// TIA Portal project "SCADA_PROJECT" (V14)

(* hardware
DEVICE "S7300/ET200M station_1"  S7-300 station
   slot 0: "Rail_0"  Rail  6ES7 390-1***0-0AA0
   slot 1: "PS 305 2A Outdoor_1"  PS 305 2A Outdoor  6ES7 305-1BA80-0AA0
   slot 2: "PLC_1"  CPU 315F-2 PN/DP  6ES7 315-2FJ14-0AB0  V3.2
      slot 2: "PROFINET interface_1"  PN-IO
         slot 1: "Port_1"  Port
         slot 2: "Port_2"  Port
   slot 4: "AI 8x12BIT_1"  AI8 x 12 bits  6ES7 331-7KF02-0AB0
   slot 5: "DO 32x24VDC/0.5A_1"  DO32 x 24VDC / 0.5A  6ES7 322-1BL00-0AA0
   slot 6: "DI 16x24VDC_1"  DI16 x 24VDC  6ES7 321-1BH50-0AA0
DEVICE "PC-System_1"  SIMATIC PC station
   slot 0: "SIMATIC PC station"  Rail  SIMATIC PC-Station  V1.0
      slot 125: "Stationmanager"  Station_Manager  V6.0.4
   slot 1: "HMI_RT_1"  WinCC RT Advanced  6AV2 104-0xxxx-xxxx  14.0.0.0
      slot 33792: "Host interface"  Host interface
   slot 2: "IE general_1"  IE General  IE_CP  V8.2.0
*)

// ===== PLC "PLC_1"  CPU 315F-2 PN/DP =====

VAR_GLOBAL   // PLC tag table "Default tag table"
   "LT1401" AT %IW256 : Int;   // Level transmitter for TANK140
   "LT1501" AT %IW258 : Int;   // Level transmitter for TANK150
   "LT1601" AT %IW260 : Int;   // Level transmitter for TANK160
   "LT1701" AT %IW262 : Int;   // Level transmitter for TANK170
   "Pump100A _start" AT %M0.0 : Bool;
   "Pump100A _stop" AT %M0.1 : Bool;
   "Pump770A _start" AT %M0.2 : Bool;
   "Pump770A_stop" AT %M0.3 : Bool;
   "Pump771A _start" AT %M0.4 : Bool;
   "Pump771A _stop" AT %M0.5 : Bool;
   "Pump100A" AT %Q4.0 : Bool;   // Status of Pump 100A
   "Pump770A" AT %Q4.1 : Bool;   // Status of Pump 770A
   "Pump771A" AT %Q4.2 : Bool;   // Status of Pump 771A
   "SV1401_open" AT %M0.6 : Bool;
   "SV1401_close" AT %M0.7 : Bool;
   "SV1501_open" AT %M1.0 : Bool;
   "SV1501_close" AT %M1.1 : Bool;
   "SV1601_open" AT %M1.2 : Bool;
   "SV1601_close" AT %M1.3 : Bool;
   "SV1701_open" AT %M1.4 : Bool;
   "SV1701_close" AT %M1.5 : Bool;
   "SV1402_open" AT %M1.6 : Bool;
   "SV1402_ close" AT %M1.7 : Bool;
   "SV1502_open" AT %M2.0 : Bool;
   "SV1502_close" AT %M2.1 : Bool;
   "SV1602_open" AT %M2.2 : Bool;
   "SV1602_ close" AT %M2.3 : Bool;
   "SV1702_open" AT %M2.4 : Bool;
   "SV1702_close" AT %M2.5 : Bool;
   "SV1401" AT %Q4.3 : Bool;   // Status of SV 1401
   "SV1501" AT %Q4.4 : Bool;   // Status of SV 1501
   "SV1601" AT %Q4.5 : Bool;   // Status of SV 1601
   "SV1701" AT %Q4.6 : Bool;   // Status of SV 1701
   "SV1402" AT %Q4.7 : Bool;   // Status of SV 1402
   "SV1502" AT %Q5.0 : Bool;   // Status of SV 1502
   "SV1602" AT %Q5.1 : Bool;   // Status of SV 1602
   "SV1702" AT %Q5.2 : Bool;   // Status of SV 1702
   "H_alarm_140" AT %Q5.3 : Bool;
   "L_alarm_140" AT %Q5.4 : Bool;
   "H_alarm_150" AT %Q5.5 : Bool;
   "L_alarm_150" AT %Q5.6 : Bool;
   "H_alarm_160" AT %Q5.7 : Bool;
   "L_alarm_160" AT %Q6.0 : Bool;
   "H_alarm_170" AT %Q6.1 : Bool;
   "L_alarm_170" AT %Q6.2 : Bool;
   "Level_real_140" AT %MD6 : Real;   // Analog value for level in Tank 140
   "Level_real_150" AT %MD10 : Real;   // Analog value for level in Tank 150
   "Level_real_160" AT %MD14 : Real;   // Analog value for level in Tank 160
   "Level_real_170" AT %MD18 : Real;   // Analog value for level in Tank 170
   "Tag_2" AT %M3.0 : Bool;   // LT140 incoming alarm
   "Tag_3" AT %M3.1 : Bool;   // LT140 out of alarm
   "Tag_4" AT %M3.2 : Bool;   // LT150 incoming alarm
   "Tag_6" AT %M3.4 : Bool;   // Pump 771A incoming alarm
   "Tag_8" AT %M3.6 : Bool;   // Pump 771A out of alarm
   "Tag_7" AT %M3.5 : Bool;   // SV1401 incoming alarm
   "Tag_9" AT %M3.7 : Bool;   // SV1401 out of alarm
   "Tag_5" AT %M3.3 : Bool;   // LT140 out of alarm
END_VAR

VAR_GLOBAL CONSTANT   // PLC tag table "Default tag table"
   "MAX_level_140" : Real := 1500.0;
   "MIN_level_140" : Real := 0.0;
   "HIGH_level_140" : Real := 1350.0;
   "LOW_level_140" : Real := 200.0;
   "MAX_level_150" : Real := 2500.0;
   "MIN_level_150" : Real := 0.0;
   "HIGH_level_150" : Real := 2250.0;
   "LOW_level_150" : Real := 200.0;
   "MAX_level_160" : Real := 3000.0;
   "MIN_level_160" : Real := 0.0;
   "HIGH_level_160" : Real := 2700.0;
   "LOW_level_160" : Real := 200.0;
   "MAX_level_170" : Real := 10000.0;
   "MIN_level_170" : Real := 0.0;
   "HIGH_level_170" : Real := 9000.0;
   "LOW_level_170" : Real := 1000.0;
END_VAR

DATA_BLOCK "FP_Database"   // DB1
{ S7_Optimized_Access := 'FALSE' }
VERSION : 0.1
   VAR
      Pump_visibility_1 : Bool := false;
      Pump100A : String := 'Pump100A';
      Pump_visibility_2 : Bool := false;
      Pump770 : String := 'Pump770';
      Pump_visibility_3 : Bool := false;
      Pump771 : String := 'Pump771';
      V_vis_1401 : Bool := false;
      "SV 1401" : String := 'SV 1401';
      V_vis_1501 : Bool := false;
      SV1501 : String := 'SV 1501';
      V_vis_1601 : Bool := false;
      SV1601 : String := 'SV 1601';
      V_vis_1701 : Bool := false;
      SV1701 : String := 'SV 1701';
      V_vis_1402 : Bool := false;
      SV1402 : String := 'SV 1402';
      V_vis_1502 : Bool := false;
      SV1502 : String := 'SV 1502';
      V_vis_1602 : Bool := false;
      SV1602 : String := 'SV 1602';
      V_vis_1702 : Bool := false;
      SV1702 : String := 'SV 1702';
   END_VAR
BEGIN
END_DATA_BLOCK

DATA_BLOCK "Alarm_DB"   // DB2
{ S7_Optimized_Access := 'FALSE' }
VERSION : 0.1
   VAR
      LT140_fault : Bool;
      LT150_fault : Bool;
      SV1401_FTC : Bool;
      SV1502_FTO : Bool;
      Pump771_FTS : Bool;
   END_VAR
BEGIN
END_DATA_BLOCK

FUNCTION "SV1x01" : Void   // FC1, LAD
{ S7_Optimized_Access := 'FALSE' }
VERSION : 0.1
   VAR_INPUT
      Open_valve : Bool;
      close_valve : Bool;
      High_alarm : Bool;
      Stop_pump : Bool;
      "Low alarm" : Bool;
   END_VAR
   VAR_OUTPUT
      SV1x01 : Bool;
   END_VAR
BEGIN

REGION Network 1
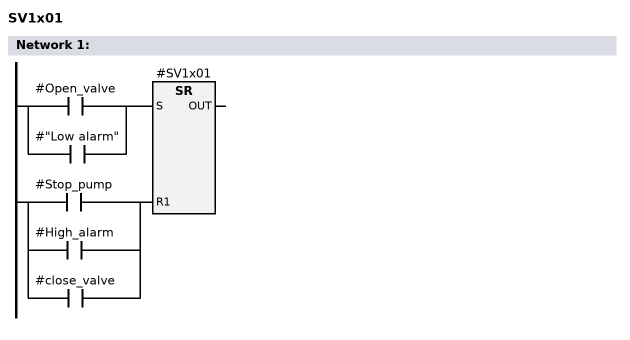
   RUNG wire#powerrail
      Contact( #Open_valve )
      wire#w1
      S_SR(operand := #SV1x01, r1 := wire#w2)
   END_RUNG
   RUNG wire#powerrail
      Contact( #"Low alarm" )
   END_RUNG wire#w1
   RUNG wire#powerrail
      Contact( #Stop_pump )
   END_RUNG wire#w2
   RUNG wire#powerrail
      Contact( #High_alarm )
   END_RUNG wire#w2
   RUNG wire#powerrail
      Contact( #close_valve )
   END_RUNG wire#w2
   // the same network as SCL:
   IF #Open_valve OR #"Low alarm" THEN
       #SV1x01 := TRUE;   // SR flip-flop
   END_IF;
   IF #Stop_pump OR #High_alarm OR #close_valve THEN #SV1x01 := FALSE; END_IF;
END_REGION
END_FUNCTION

FUNCTION "Tank_Alarm" : Void   // FC2, LAD
{ S7_Optimized_Access := 'FALSE' }
VERSION : 0.1
   VAR_INPUT
      LT1x01 : Int;
      High_Level : Real;
      Low_Level : Real;
      HIGH_alarm_limit : Real;
      LOW_alarm_limit : Real;
   END_VAR
   VAR_OUTPUT
      High_alarm : Bool;
      Low_alarm : Bool;
   END_VAR
   VAR_IN_OUT
      Level : Real;
   END_VAR
   VAR_TEMP
      Bipolar : Bool;
      Value : Word;
   END_VAR
BEGIN

REGION Network 1
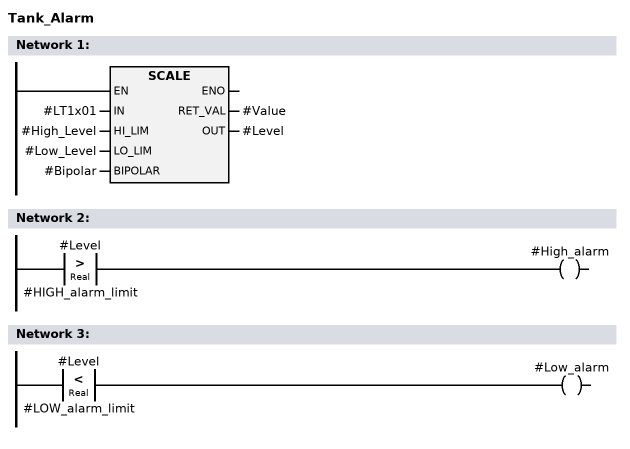
   #Value := SCALE(IN := #LT1x01,
                   HI_LIM := #High_Level,
                   LO_LIM := #Low_Level,
                   BIPOLAR := #Bipolar,
                   OUT => #Level);
END_REGION

REGION Network 2
   RUNG wire#powerrail
      { S7_Templates := "SrcType := Real" } GT_Contact(in1 := #Level, in2 := #HIGH_alarm_limit)
      Coil( #High_alarm )
   END_RUNG
   // the same network as SCL:
   #High_alarm := #Level > #HIGH_alarm_limit;
END_REGION

REGION Network 3
   RUNG wire#powerrail
      { S7_Templates := "SrcType := Real" } LT_Contact(in1 := #Level, in2 := #LOW_alarm_limit)
      Coil( #Low_alarm )
   END_RUNG
   // the same network as SCL:
   #Low_alarm := #Level < #LOW_alarm_limit;
END_REGION
END_FUNCTION

FUNCTION "PUMP_100A" : Void   // FC3, LAD
{ S7_Optimized_Access := 'FALSE' }
VERSION : 0.1
   VAR_INPUT
      SV1x01_1 : Bool;
      SVx01_2 : Bool;
      SV1x01_3 : Bool;
      START_PUMP : Bool;
      STOP_PUMP : Bool;
      Pump770A : Bool;
      SV1701 : Bool;
      L_140 : Bool;
      L_150 : Bool;
      L_160 : Bool;
   END_VAR
   VAR_OUTPUT
      PUMP100A : Bool;
   END_VAR
BEGIN

REGION Network 1
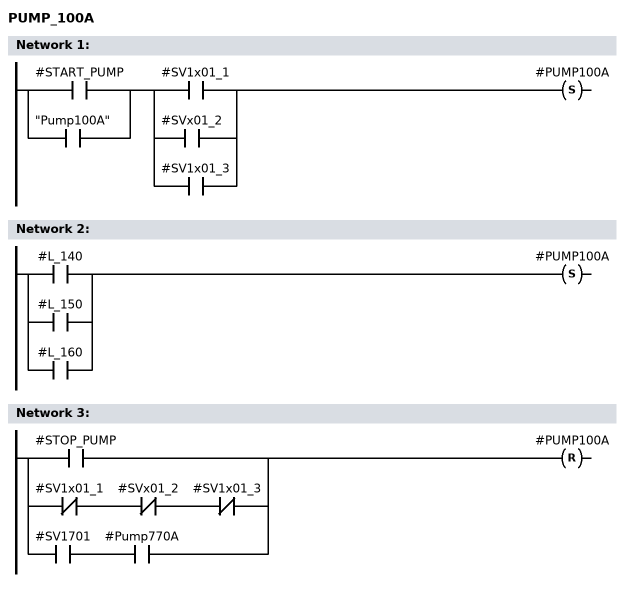
   RUNG wire#powerrail
      Contact( #START_PUMP )
      wire#w1
      Contact( #SV1x01_1 )
      wire#w2
      S_Coil( #PUMP100A )
   END_RUNG
   RUNG wire#powerrail
      Contact( "Pump100A" )
   END_RUNG wire#w1
   RUNG wire#w1
      Contact( #SVx01_2 )
   END_RUNG wire#w2
   RUNG wire#w1
      Contact( #SV1x01_3 )
   END_RUNG wire#w2
   // the same network as SCL:
   IF (#START_PUMP OR "Pump100A") AND (#SV1x01_1 OR #SVx01_2 OR #SV1x01_3) THEN #PUMP100A := TRUE; END_IF;
END_REGION

REGION Network 2
   RUNG wire#powerrail
      Contact( #L_140 )
      wire#w1
      S_Coil( #PUMP100A )
   END_RUNG
   RUNG wire#powerrail
      Contact( #L_150 )
   END_RUNG wire#w1
   RUNG wire#powerrail
      Contact( #L_160 )
   END_RUNG wire#w1
   // the same network as SCL:
   IF #L_140 OR #L_150 OR #L_160 THEN #PUMP100A := TRUE; END_IF;
END_REGION

REGION Network 3
   RUNG wire#powerrail
      Contact( #STOP_PUMP )
      wire#w1
      R_Coil( #PUMP100A )
   END_RUNG
   RUNG wire#powerrail
      I_Contact( #SV1x01_1 )
      I_Contact( #SVx01_2 )
      I_Contact( #SV1x01_3 )
   END_RUNG wire#w1
   RUNG wire#powerrail
      Contact( #SV1701 )
      Contact( #Pump770A )
   END_RUNG wire#w1
   // the same network as SCL:
   IF #STOP_PUMP OR (NOT #SV1x01_1 AND NOT #SVx01_2 AND NOT #SV1x01_3) OR (#SV1701 AND #Pump770A) THEN
       #PUMP100A := FALSE;
   END_IF;
END_REGION
END_FUNCTION

FUNCTION "SV1x02" : Void   // FC4, LAD
{ S7_Optimized_Access := 'FALSE' }
VERSION : 0.1
   VAR_INPUT
      Open_valve : Bool;
      SV1x01 : Bool;
      Low_alarm_170 : Bool;
      High_Alarm : Bool;
      Low_alarm : Bool;
      High_alarm_170 : Bool;
      close_valve : Bool;
      Pump100A : Bool;
   END_VAR
   VAR_OUTPUT
      SV_1x02 : Bool;
   END_VAR
BEGIN

REGION Network 1
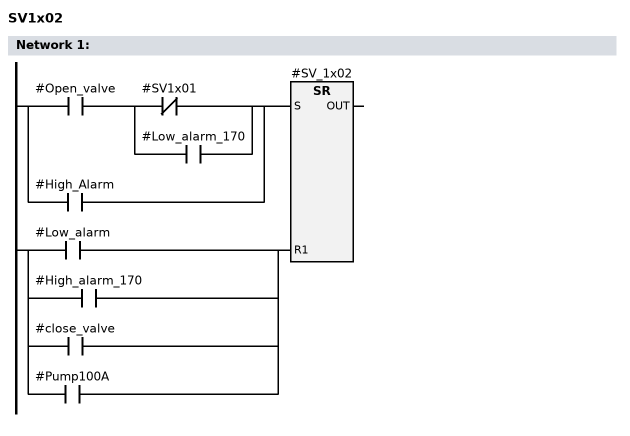
   RUNG wire#powerrail
      Contact( #Open_valve )
      wire#w1
      I_Contact( #SV1x01 )
      wire#w2
      S_SR(operand := #SV_1x02, r1 := wire#w3)
   END_RUNG
   RUNG wire#w1
      Contact( #Low_alarm_170 )
   END_RUNG wire#w2
   RUNG wire#powerrail
      Contact( #High_Alarm )
   END_RUNG wire#w2
   RUNG wire#powerrail
      Contact( #Low_alarm )
   END_RUNG wire#w3
   RUNG wire#powerrail
      Contact( #High_alarm_170 )
   END_RUNG wire#w3
   RUNG wire#powerrail
      Contact( #close_valve )
   END_RUNG wire#w3
   RUNG wire#powerrail
      Contact( #Pump100A )
   END_RUNG wire#w3
   // the same network as SCL:
   IF (#Open_valve AND (NOT #SV1x01 OR #Low_alarm_170)) OR #High_Alarm THEN
       #SV_1x02 := TRUE;   // SR flip-flop
   END_IF;
   IF #Low_alarm OR #High_alarm_170 OR #close_valve OR #Pump100A THEN #SV_1x02 := FALSE; END_IF;
END_REGION
END_FUNCTION

FUNCTION "SV_1702" : Void   // FC6, LAD
{ S7_Optimized_Access := 'FALSE' }
VERSION : 0.1
   VAR_INPUT
      Open_valve : Bool;
      High_170 : Bool;
      Close_valve : Bool;
      LOW_170 : Bool;
      SV1701 : Bool;
      PUMP770A : Bool;
   END_VAR
   VAR_OUTPUT
      SV_1702 : Bool;
   END_VAR
BEGIN

REGION Network 1
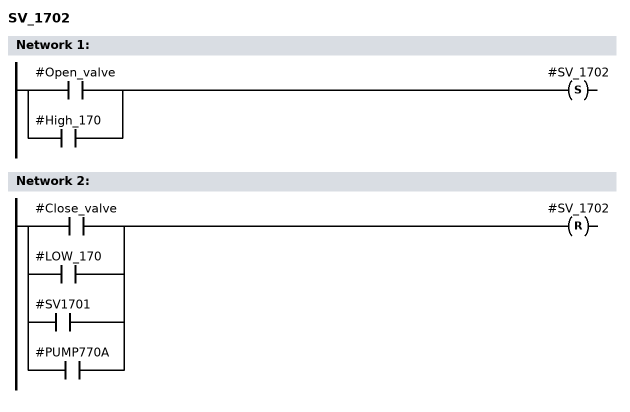
   RUNG wire#powerrail
      Contact( #Open_valve )
      wire#w1
      S_Coil( #SV_1702 )
   END_RUNG
   RUNG wire#powerrail
      Contact( #High_170 )
   END_RUNG wire#w1
   // the same network as SCL:
   IF #Open_valve OR #High_170 THEN #SV_1702 := TRUE; END_IF;
END_REGION

REGION Network 2
   RUNG wire#powerrail
      Contact( #Close_valve )
      wire#w1
      R_Coil( #SV_1702 )
   END_RUNG
   RUNG wire#powerrail
      Contact( #LOW_170 )
   END_RUNG wire#w1
   RUNG wire#powerrail
      Contact( #SV1701 )
   END_RUNG wire#w1
   RUNG wire#powerrail
      Contact( #PUMP770A )
   END_RUNG wire#w1
   // the same network as SCL:
   IF #Close_valve OR #LOW_170 OR #SV1701 OR #PUMP770A THEN #SV_1702 := FALSE; END_IF;
END_REGION
END_FUNCTION

FUNCTION "PUMP_770A" : Void   // FC7, LAD
{ S7_Optimized_Access := 'FALSE' }
VERSION : 0.1
   VAR_INPUT
      Start_pump : Bool;
      SV1701 : Bool;
      Low170 : Bool;
      Stop_pump : Bool;
      High170 : Bool;
      SV1x02_1 : Bool;
      SVx02_2 : Bool;
      SV1x02_3 : Bool;
      SV1702 : Bool;
      "PUMP _771A" : Bool;
      PUMP_100A : Bool;
   END_VAR
   VAR_OUTPUT
      Pump770 : Bool;
   END_VAR
BEGIN

REGION Network 1
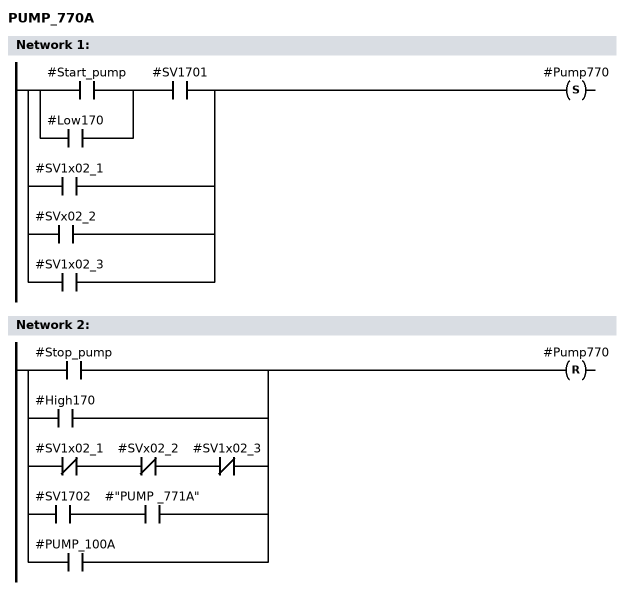
   RUNG wire#powerrail
      Contact( #Start_pump )
      wire#w1
      Contact( #SV1701 )
      wire#w2
      S_Coil( #Pump770 )
   END_RUNG
   RUNG wire#powerrail
      Contact( #Low170 )
   END_RUNG wire#w1
   RUNG wire#powerrail
      Contact( #SV1x02_1 )
   END_RUNG wire#w2
   RUNG wire#powerrail
      Contact( #SVx02_2 )
   END_RUNG wire#w2
   RUNG wire#powerrail
      Contact( #SV1x02_3 )
   END_RUNG wire#w2
   // the same network as SCL:
   IF ((#Start_pump OR #Low170) AND #SV1701) OR #SV1x02_1 OR #SVx02_2 OR #SV1x02_3 THEN
       #Pump770 := TRUE;
   END_IF;
END_REGION

REGION Network 2
   RUNG wire#powerrail
      Contact( #Stop_pump )
      wire#w1
      R_Coil( #Pump770 )
   END_RUNG
   RUNG wire#powerrail
      Contact( #High170 )
   END_RUNG wire#w1
   RUNG wire#powerrail
      I_Contact( #SV1x02_1 )
      I_Contact( #SVx02_2 )
      I_Contact( #SV1x02_3 )
   END_RUNG wire#w1
   RUNG wire#powerrail
      Contact( #SV1702 )
      Contact( #"PUMP _771A" )
   END_RUNG wire#w1
   RUNG wire#powerrail
      Contact( #PUMP_100A )
   END_RUNG wire#w1
   // the same network as SCL:
   IF #Stop_pump OR #High170 OR (NOT #SV1x02_1 AND NOT #SVx02_2 AND NOT #SV1x02_3) OR (#SV1702 AND #"PUMP _771A") OR #PUMP_100A THEN
       #Pump770 := FALSE;
   END_IF;
END_REGION
END_FUNCTION

FUNCTION "PUMP_771A" : Void   // FC8, LAD
{ S7_Optimized_Access := 'FALSE' }
VERSION : 0.1
   VAR_INPUT
      START_PUMP : Bool;
      SV1702 : Bool;
      High_170 : Bool;
      STOP_Pump : Bool;
      LOW_170 : Bool;
      SV1701 : Bool;
      Pump770A : Bool;
      Pump100A : Bool;
   END_VAR
   VAR_OUTPUT
      PUMP771A : Bool;
   END_VAR
BEGIN

REGION Network 1
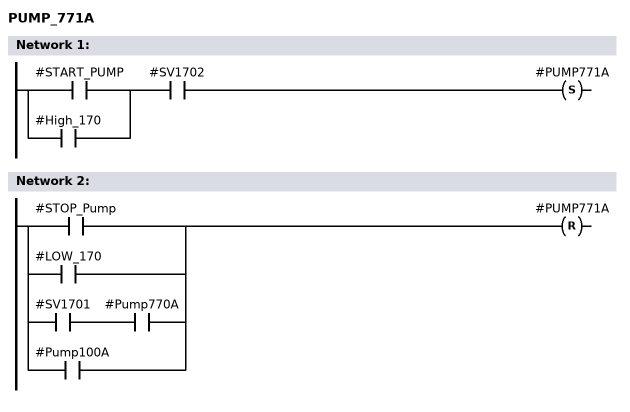
   RUNG wire#powerrail
      Contact( #START_PUMP )
      wire#w1
      Contact( #SV1702 )
      S_Coil( #PUMP771A )
   END_RUNG
   RUNG wire#powerrail
      Contact( #High_170 )
   END_RUNG wire#w1
   // the same network as SCL:
   IF (#START_PUMP OR #High_170) AND #SV1702 THEN #PUMP771A := TRUE; END_IF;
END_REGION

REGION Network 2
   RUNG wire#powerrail
      Contact( #STOP_Pump )
      wire#w1
      R_Coil( #PUMP771A )
   END_RUNG
   RUNG wire#powerrail
      Contact( #LOW_170 )
   END_RUNG wire#w1
   RUNG wire#powerrail
      Contact( #SV1701 )
      Contact( #Pump770A )
   END_RUNG wire#w1
   RUNG wire#powerrail
      Contact( #Pump100A )
   END_RUNG wire#w1
   // the same network as SCL:
   IF #STOP_Pump OR #LOW_170 OR (#SV1701 AND #Pump770A) OR #Pump100A THEN #PUMP771A := FALSE; END_IF;
END_REGION
END_FUNCTION

FUNCTION "SV_1701" : Void   // FC9, LAD
{ S7_Optimized_Access := 'FALSE' }
VERSION : 0.1
   VAR_INPUT
      OPEN_valve : Bool;
      SV1402 : Bool;
      SV1502 : Bool;
      SV1602 : Bool;
      Close_valve : Bool;
      HIGH_170 : Bool;
   END_VAR
   VAR_OUTPUT
      SV1701 : Bool;
   END_VAR
BEGIN

REGION Network 1
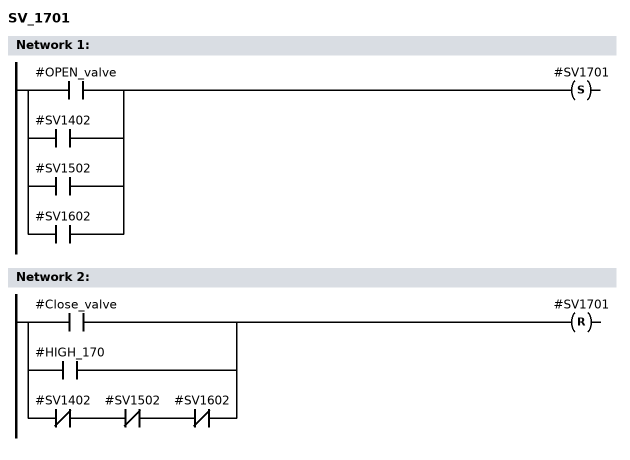
   RUNG wire#powerrail
      Contact( #OPEN_valve )
      wire#w1
      S_Coil( #SV1701 )
   END_RUNG
   RUNG wire#powerrail
      Contact( #SV1402 )
   END_RUNG wire#w1
   RUNG wire#powerrail
      Contact( #SV1502 )
   END_RUNG wire#w1
   RUNG wire#powerrail
      Contact( #SV1602 )
   END_RUNG wire#w1
   // the same network as SCL:
   IF #OPEN_valve OR #SV1402 OR #SV1502 OR #SV1602 THEN #SV1701 := TRUE; END_IF;
END_REGION

REGION Network 2
   RUNG wire#powerrail
      Contact( #Close_valve )
      wire#w1
      R_Coil( #SV1701 )
   END_RUNG
   RUNG wire#powerrail
      Contact( #HIGH_170 )
   END_RUNG wire#w1
   RUNG wire#powerrail
      I_Contact( #SV1402 )
      I_Contact( #SV1502 )
      I_Contact( #SV1602 )
   END_RUNG wire#w1
   // the same network as SCL:
   IF #Close_valve OR #HIGH_170 OR (NOT #SV1402 AND NOT #SV1502 AND NOT #SV1602) THEN
       #SV1701 := FALSE;
   END_IF;
END_REGION
END_FUNCTION

ORGANIZATION_BLOCK "Main"   // OB1, LAD
TITLE = "Main Program Sweep (Cycle)"
{ S7_Optimized_Access := 'FALSE' }
VERSION : 0.1
   VAR_TEMP
      OB1_EV_CLASS : Byte;   // Bits 0-3 = 1 (Coming event), Bits 4-7 = 1 (Event class 1)
      OB1_SCAN_1 : Byte;   // 1 (Cold restart scan 1 of OB 1), 3 (Scan 2-n of OB 1)
      OB1_PRIORITY : Byte;   // Priority of OB Execution
      OB1_OB_NUMBR : Byte;   // 1 (Organization block 1, OB1)
      OB1_RESERVED_1 : Byte;   // Reserved for system
      OB1_RESERVED_2 : Byte;   // Reserved for system
      OB1_PREV_CYCLE : Int;   // Cycle time of previous OB1 scan (milliseconds)
      OB1_MIN_CYCLE : Int;   // Minimum cycle time of OB1 (milliseconds)
      OB1_MAX_CYCLE : Int;   // Maximum cycle time of OB1 (milliseconds)
      OB1_DATE_TIME : Date_And_Time;   // Date and time OB1 started
   END_VAR
BEGIN

REGION Network 1
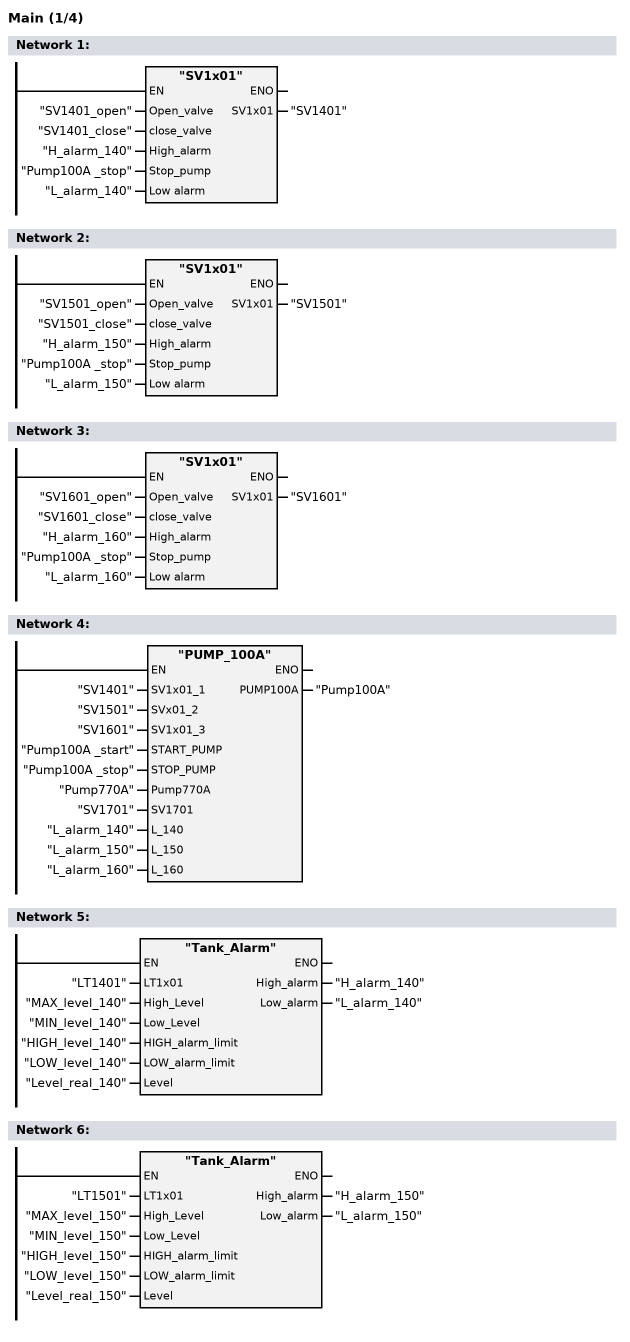
   RUNG wire#powerrail
      "SV1x01"(Open_valve := "SV1401_open", close_valve := "SV1401_close", High_alarm := "H_alarm_140", Stop_pump := "Pump100A _stop", "Low alarm" := "L_alarm_140", SV1x01 => "SV1401")
   END_RUNG
   // the same network as SCL:
   "SV1x01"(Open_valve := "SV1401_open",
            close_valve := "SV1401_close",
            High_alarm := "H_alarm_140",
            Stop_pump := "Pump100A _stop",
            "Low alarm" := "L_alarm_140",
            SV1x01 => "SV1401");
END_REGION

REGION Network 2
   RUNG wire#powerrail
      "SV1x01"(Open_valve := "SV1501_open", close_valve := "SV1501_close", High_alarm := "H_alarm_150", Stop_pump := "Pump100A _stop", "Low alarm" := "L_alarm_150", SV1x01 => "SV1501")
   END_RUNG
   // the same network as SCL:
   "SV1x01"(Open_valve := "SV1501_open",
            close_valve := "SV1501_close",
            High_alarm := "H_alarm_150",
            Stop_pump := "Pump100A _stop",
            "Low alarm" := "L_alarm_150",
            SV1x01 => "SV1501");
END_REGION

REGION Network 3
   RUNG wire#powerrail
      "SV1x01"(Open_valve := "SV1601_open", close_valve := "SV1601_close", High_alarm := "H_alarm_160", Stop_pump := "Pump100A _stop", "Low alarm" := "L_alarm_160", SV1x01 => "SV1601")
   END_RUNG
   // the same network as SCL:
   "SV1x01"(Open_valve := "SV1601_open",
            close_valve := "SV1601_close",
            High_alarm := "H_alarm_160",
            Stop_pump := "Pump100A _stop",
            "Low alarm" := "L_alarm_160",
            SV1x01 => "SV1601");
END_REGION

REGION Network 4
   RUNG wire#powerrail
      "PUMP_100A"(SV1x01_1 := "SV1401", SVx01_2 := "SV1501", SV1x01_3 := "SV1601", START_PUMP := "Pump100A _start", STOP_PUMP := "Pump100A _stop", Pump770A := "Pump770A", SV1701 := "SV1701", L_140 := "L_alarm_140", L_150 := "L_alarm_150", L_160 := "L_alarm_160", PUMP100A => "Pump100A")
   END_RUNG
   // the same network as SCL:
   "PUMP_100A"(SV1x01_1 := "SV1401",
               SVx01_2 := "SV1501",
               SV1x01_3 := "SV1601",
               START_PUMP := "Pump100A _start",
               STOP_PUMP := "Pump100A _stop",
               Pump770A := "Pump770A",
               SV1701 := "SV1701",
               L_140 := "L_alarm_140",
               L_150 := "L_alarm_150",
               L_160 := "L_alarm_160",
               PUMP100A => "Pump100A");
END_REGION

REGION Network 5
   RUNG wire#powerrail
      "Tank_Alarm"(LT1x01 := "LT1401", High_Level := "MAX_level_140", Low_Level := "MIN_level_140", HIGH_alarm_limit := "HIGH_level_140", LOW_alarm_limit := "LOW_level_140", Level := "Level_real_140", High_alarm => "H_alarm_140", Low_alarm => "L_alarm_140")
   END_RUNG
   // the same network as SCL:
   "Tank_Alarm"(LT1x01 := "LT1401",
                High_Level := "MAX_level_140",
                Low_Level := "MIN_level_140",
                HIGH_alarm_limit := "HIGH_level_140",
                LOW_alarm_limit := "LOW_level_140",
                Level := "Level_real_140",
                High_alarm => "H_alarm_140",
                Low_alarm => "L_alarm_140");
END_REGION

REGION Network 6
   RUNG wire#powerrail
      "Tank_Alarm"(LT1x01 := "LT1501", High_Level := "MAX_level_150", Low_Level := "MIN_level_150", HIGH_alarm_limit := "HIGH_level_150", LOW_alarm_limit := "LOW_level_150", Level := "Level_real_150", High_alarm => "H_alarm_150", Low_alarm => "L_alarm_150")
   END_RUNG
   // the same network as SCL:
   "Tank_Alarm"(LT1x01 := "LT1501",
                High_Level := "MAX_level_150",
                Low_Level := "MIN_level_150",
                HIGH_alarm_limit := "HIGH_level_150",
                LOW_alarm_limit := "LOW_level_150",
                Level := "Level_real_150",
                High_alarm => "H_alarm_150",
                Low_alarm => "L_alarm_150");
END_REGION

REGION Network 7
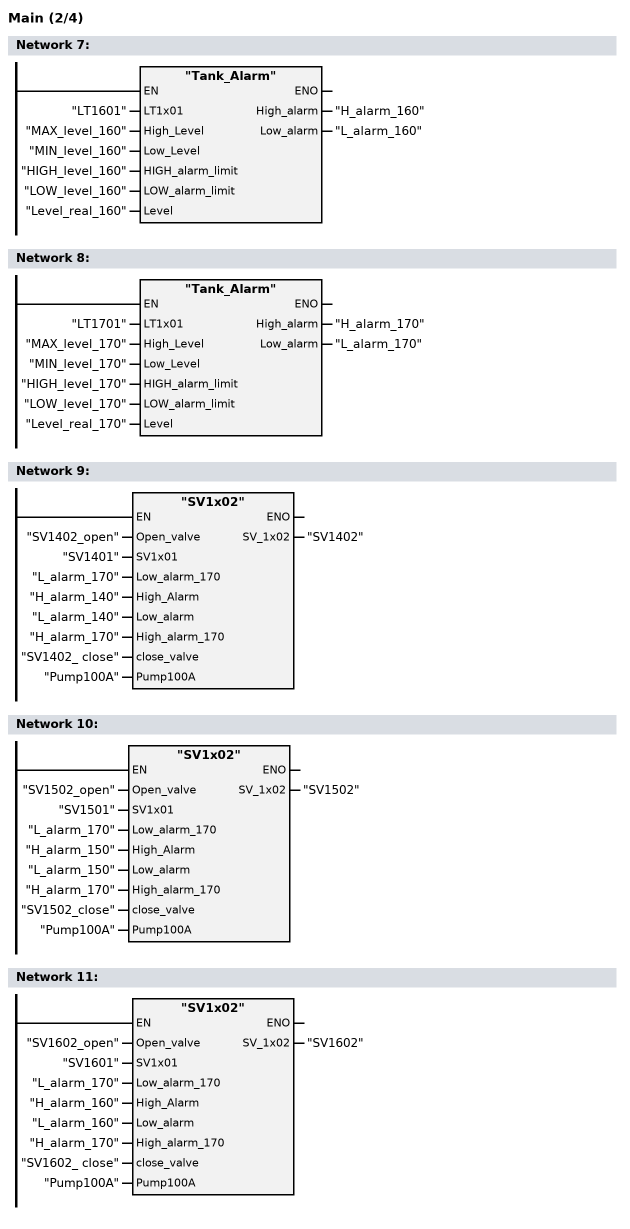
   RUNG wire#powerrail
      "Tank_Alarm"(LT1x01 := "LT1601", High_Level := "MAX_level_160", Low_Level := "MIN_level_160", HIGH_alarm_limit := "HIGH_level_160", LOW_alarm_limit := "LOW_level_160", Level := "Level_real_160", High_alarm => "H_alarm_160", Low_alarm => "L_alarm_160")
   END_RUNG
   // the same network as SCL:
   "Tank_Alarm"(LT1x01 := "LT1601",
                High_Level := "MAX_level_160",
                Low_Level := "MIN_level_160",
                HIGH_alarm_limit := "HIGH_level_160",
                LOW_alarm_limit := "LOW_level_160",
                Level := "Level_real_160",
                High_alarm => "H_alarm_160",
                Low_alarm => "L_alarm_160");
END_REGION

REGION Network 8
   RUNG wire#powerrail
      "Tank_Alarm"(LT1x01 := "LT1701", High_Level := "MAX_level_170", Low_Level := "MIN_level_170", HIGH_alarm_limit := "HIGH_level_170", LOW_alarm_limit := "LOW_level_170", Level := "Level_real_170", High_alarm => "H_alarm_170", Low_alarm => "L_alarm_170")
   END_RUNG
   // the same network as SCL:
   "Tank_Alarm"(LT1x01 := "LT1701",
                High_Level := "MAX_level_170",
                Low_Level := "MIN_level_170",
                HIGH_alarm_limit := "HIGH_level_170",
                LOW_alarm_limit := "LOW_level_170",
                Level := "Level_real_170",
                High_alarm => "H_alarm_170",
                Low_alarm => "L_alarm_170");
END_REGION

REGION Network 9
   RUNG wire#powerrail
      "SV1x02"(Open_valve := "SV1402_open", SV1x01 := "SV1401", Low_alarm_170 := "L_alarm_170", High_Alarm := "H_alarm_140", Low_alarm := "L_alarm_140", High_alarm_170 := "H_alarm_170", close_valve := "SV1402_ close", Pump100A := "Pump100A", SV_1x02 => "SV1402")
   END_RUNG
   // the same network as SCL:
   "SV1x02"(Open_valve := "SV1402_open",
            SV1x01 := "SV1401",
            Low_alarm_170 := "L_alarm_170",
            High_Alarm := "H_alarm_140",
            Low_alarm := "L_alarm_140",
            High_alarm_170 := "H_alarm_170",
            close_valve := "SV1402_ close",
            Pump100A := "Pump100A",
            SV_1x02 => "SV1402");
END_REGION

REGION Network 10
   RUNG wire#powerrail
      "SV1x02"(Open_valve := "SV1502_open", SV1x01 := "SV1501", Low_alarm_170 := "L_alarm_170", High_Alarm := "H_alarm_150", Low_alarm := "L_alarm_150", High_alarm_170 := "H_alarm_170", close_valve := "SV1502_close", Pump100A := "Pump100A", SV_1x02 => "SV1502")
   END_RUNG
   // the same network as SCL:
   "SV1x02"(Open_valve := "SV1502_open",
            SV1x01 := "SV1501",
            Low_alarm_170 := "L_alarm_170",
            High_Alarm := "H_alarm_150",
            Low_alarm := "L_alarm_150",
            High_alarm_170 := "H_alarm_170",
            close_valve := "SV1502_close",
            Pump100A := "Pump100A",
            SV_1x02 => "SV1502");
END_REGION

REGION Network 11
   RUNG wire#powerrail
      "SV1x02"(Open_valve := "SV1602_open", SV1x01 := "SV1601", Low_alarm_170 := "L_alarm_170", High_Alarm := "H_alarm_160", Low_alarm := "L_alarm_160", High_alarm_170 := "H_alarm_170", close_valve := "SV1602_ close", Pump100A := "Pump100A", SV_1x02 => "SV1602")
   END_RUNG
   // the same network as SCL:
   "SV1x02"(Open_valve := "SV1602_open",
            SV1x01 := "SV1601",
            Low_alarm_170 := "L_alarm_170",
            High_Alarm := "H_alarm_160",
            Low_alarm := "L_alarm_160",
            High_alarm_170 := "H_alarm_170",
            close_valve := "SV1602_ close",
            Pump100A := "Pump100A",
            SV_1x02 => "SV1602");
END_REGION

REGION Network 12
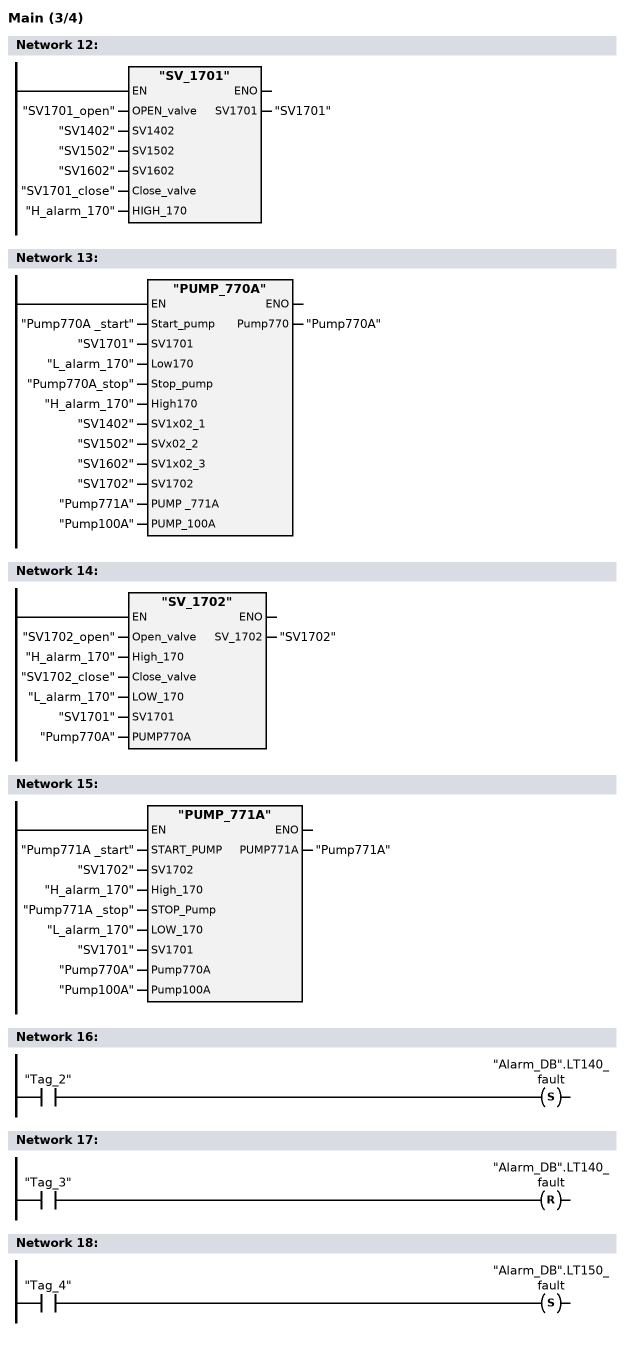
   RUNG wire#powerrail
      "SV_1701"(OPEN_valve := "SV1701_open", SV1402 := "SV1402", SV1502 := "SV1502", SV1602 := "SV1602", Close_valve := "SV1701_close", HIGH_170 := "H_alarm_170", SV1701 => "SV1701")
   END_RUNG
   // the same network as SCL:
   "SV_1701"(OPEN_valve := "SV1701_open",
             SV1402 := "SV1402",
             SV1502 := "SV1502",
             SV1602 := "SV1602",
             Close_valve := "SV1701_close",
             HIGH_170 := "H_alarm_170",
             SV1701 => "SV1701");
END_REGION

REGION Network 13
   RUNG wire#powerrail
      "PUMP_770A"(Start_pump := "Pump770A _start", SV1701 := "SV1701", Low170 := "L_alarm_170", Stop_pump := "Pump770A_stop", High170 := "H_alarm_170", SV1x02_1 := "SV1402", SVx02_2 := "SV1502", SV1x02_3 := "SV1602", SV1702 := "SV1702", "PUMP _771A" := "Pump771A", PUMP_100A := "Pump100A", Pump770 => "Pump770A")
   END_RUNG
   // the same network as SCL:
   "PUMP_770A"(Start_pump := "Pump770A _start",
               SV1701 := "SV1701",
               Low170 := "L_alarm_170",
               Stop_pump := "Pump770A_stop",
               High170 := "H_alarm_170",
               SV1x02_1 := "SV1402",
               SVx02_2 := "SV1502",
               SV1x02_3 := "SV1602",
               SV1702 := "SV1702",
               "PUMP _771A" := "Pump771A",
               PUMP_100A := "Pump100A",
               Pump770 => "Pump770A");
END_REGION

REGION Network 14
   RUNG wire#powerrail
      "SV_1702"(Open_valve := "SV1702_open", High_170 := "H_alarm_170", Close_valve := "SV1702_close", LOW_170 := "L_alarm_170", SV1701 := "SV1701", PUMP770A := "Pump770A", SV_1702 => "SV1702")
   END_RUNG
   // the same network as SCL:
   "SV_1702"(Open_valve := "SV1702_open",
             High_170 := "H_alarm_170",
             Close_valve := "SV1702_close",
             LOW_170 := "L_alarm_170",
             SV1701 := "SV1701",
             PUMP770A := "Pump770A",
             SV_1702 => "SV1702");
END_REGION

REGION Network 15
   RUNG wire#powerrail
      "PUMP_771A"(START_PUMP := "Pump771A _start", SV1702 := "SV1702", High_170 := "H_alarm_170", STOP_Pump := "Pump771A _stop", LOW_170 := "L_alarm_170", SV1701 := "SV1701", Pump770A := "Pump770A", Pump100A := "Pump100A", PUMP771A => "Pump771A")
   END_RUNG
   // the same network as SCL:
   "PUMP_771A"(START_PUMP := "Pump771A _start",
               SV1702 := "SV1702",
               High_170 := "H_alarm_170",
               STOP_Pump := "Pump771A _stop",
               LOW_170 := "L_alarm_170",
               SV1701 := "SV1701",
               Pump770A := "Pump770A",
               Pump100A := "Pump100A",
               PUMP771A => "Pump771A");
END_REGION

REGION Network 16
   RUNG wire#powerrail
      Contact( "Tag_2" )
      S_Coil( "Alarm_DB".LT140_fault )
   END_RUNG
   // the same network as SCL:
   IF "Tag_2" THEN "Alarm_DB".LT140_fault := TRUE; END_IF;
END_REGION

REGION Network 17
   RUNG wire#powerrail
      Contact( "Tag_3" )
      R_Coil( "Alarm_DB".LT140_fault )
   END_RUNG
   // the same network as SCL:
   IF "Tag_3" THEN "Alarm_DB".LT140_fault := FALSE; END_IF;
END_REGION

REGION Network 18
   RUNG wire#powerrail
      Contact( "Tag_4" )
      S_Coil( "Alarm_DB".LT150_fault )
   END_RUNG
   // the same network as SCL:
   IF "Tag_4" THEN "Alarm_DB".LT150_fault := TRUE; END_IF;
END_REGION

REGION Network 19
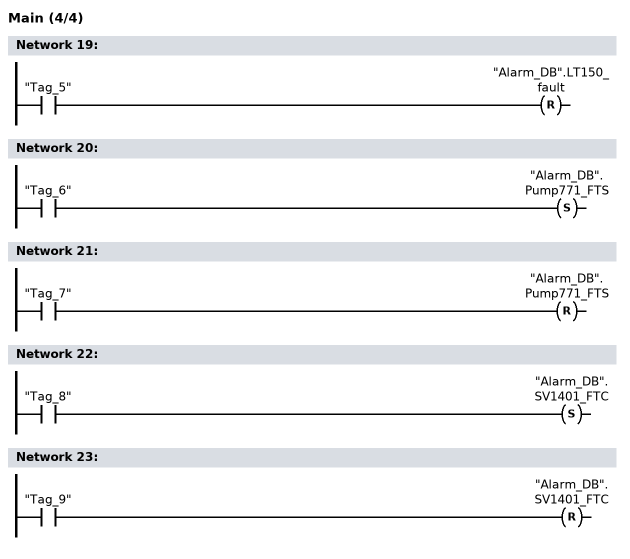
   RUNG wire#powerrail
      Contact( "Tag_5" )
      R_Coil( "Alarm_DB".LT150_fault )
   END_RUNG
   // the same network as SCL:
   IF "Tag_5" THEN "Alarm_DB".LT150_fault := FALSE; END_IF;
END_REGION

REGION Network 20
   RUNG wire#powerrail
      Contact( "Tag_6" )
      S_Coil( "Alarm_DB".Pump771_FTS )
   END_RUNG
   // the same network as SCL:
   IF "Tag_6" THEN "Alarm_DB".Pump771_FTS := TRUE; END_IF;
END_REGION

REGION Network 21
   RUNG wire#powerrail
      Contact( "Tag_7" )
      R_Coil( "Alarm_DB".Pump771_FTS )
   END_RUNG
   // the same network as SCL:
   IF "Tag_7" THEN "Alarm_DB".Pump771_FTS := FALSE; END_IF;
END_REGION

REGION Network 22
   RUNG wire#powerrail
      Contact( "Tag_8" )
      S_Coil( "Alarm_DB".SV1401_FTC )
   END_RUNG
   // the same network as SCL:
   IF "Tag_8" THEN "Alarm_DB".SV1401_FTC := TRUE; END_IF;
END_REGION

REGION Network 23
   RUNG wire#powerrail
      Contact( "Tag_9" )
      R_Coil( "Alarm_DB".SV1401_FTC )
   END_RUNG
   // the same network as SCL:
   IF "Tag_9" THEN "Alarm_DB".SV1401_FTC := FALSE; END_IF;
END_REGION
END_ORGANIZATION_BLOCK

(* ===== HMI "HMI_RT_1" =====
system functions are stored by id; their names below are inferred from use
connection "HMI_Connection_1": ETHERNET, SIMATIC S7 300/400 MPI

HMI tags "Default tag table"
   "Current_user" : WString[10], internal
   "Gruop_number" : Int, internal
   "H_alarm_140" : Bool = PLC H_alarm_140 AT %Q5.3, 1 s
   "L_alarm_140" : Bool = PLC L_alarm_140 AT %Q5.4, 1 s
   "SV1401" : Bool = PLC SV1401 AT %Q4.3, 1 s
   "Pump100A" : Bool = PLC Pump100A AT %Q4.0, 1 s
   "SV1402" : Bool = PLC SV1402 AT %Q4.7, 1 s
   "H_alarm_150" : Bool = PLC H_alarm_150 AT %Q5.5, 1 s
   "L_alarm_150" : Bool = PLC L_alarm_150 AT %Q5.6, 1 s
   "L_alarm_160" : Bool = PLC L_alarm_160 AT %Q6.0, 1 s
   "H_alarm_160" : Bool = PLC H_alarm_160 AT %Q5.7, 1 s
   "SV1501" : Bool = PLC SV1501 AT %Q4.4, 1 s
   "SV1502" : Bool = PLC SV1502 AT %Q5.0, 1 s
   "SV1601" : Bool = PLC SV1601 AT %Q4.5, 1 s
   "SV1602" : Bool = PLC SV1602 AT %Q5.1, 1 s
   "Pump770A" : Bool = PLC Pump770A AT %Q4.1, 1 s
   "Pump771A" : Bool = PLC Pump771A AT %Q4.2, 1 s
   "Pump100A _start" : Bool = PLC "Pump100A _start" AT %M0.0, 1 s
   "Pump100A _stop" : Bool = PLC "Pump100A _stop" AT %M0.1, 1 s
   "FP_Database_Pump100A" : String[254] = PLC FP_Database.Pump100A AT %DB1.DBX2.0, 1 s
   "FP_Database_Pump_visibility_2" : Bool = PLC FP_Database.Pump_visibility_2 AT %DB1.DBX258.0, 1 s
   "FP_Database_Pump_visibility_3" : Bool = PLC FP_Database.Pump_visibility_3 AT %DB1.DBX516.0, 1 s
   "Pump770A _start" : Bool = PLC "Pump770A _start" AT %M0.2, 1 s
   "Pump770A_stop" : Bool = PLC Pump770A_stop AT %M0.3, 1 s
   "FP_Database_Pump770" : String[254] = PLC FP_Database.Pump770 AT %DB1.DBX260.0, 1 s
   "Pump771A _start" : Bool = PLC "Pump771A _start" AT %M0.4, 1 s
   "Pump771A _stop" : Bool = PLC "Pump771A _stop" AT %M0.5, 1 s
   "FP_Database_Pump771" : String[254] = PLC FP_Database.Pump771 AT %DB1.DBX518.0, 1 s
   "SV1702" : Bool = PLC SV1702 AT %Q5.2, 1 s
   "H_alarm_170" : Bool = PLC H_alarm_170 AT %Q6.1, 1 s
   "L_alarm_170" : Bool = PLC L_alarm_170 AT %Q6.2, 1 s
   "FP_Database_V_vis_1401" : Bool = PLC FP_Database.V_vis_1401 AT %DB1.DBX774.0, 1 s
   "FP_Database_V_vis_1402" : Bool = PLC FP_Database.V_vis_1402 AT %DB1.DBX1806.0, 1 s
   "FP_Database_V_vis_1501" : Bool = PLC FP_Database.V_vis_1501 AT %DB1.DBX1032.0, 1 s
   "FP_Database_V_vis_1502" : Bool = PLC FP_Database.V_vis_1502 AT %DB1.DBX2064.0, 1 s
   "FP_Database_V_vis_1601" : Bool = PLC FP_Database.V_vis_1601 AT %DB1.DBX1290.0, 1 s
   "FP_Database_V_vis_1602" : Bool = PLC FP_Database.V_vis_1602 AT %DB1.DBX2322.0, 1 s
   "FP_Database_V_vis_1701" : Bool = PLC FP_Database.V_vis_1701 AT %DB1.DBX1548.0, 1 s
   "FP_Database_V_vis_1702" : Bool = PLC FP_Database.V_vis_1702 AT %DB1.DBX2580.0, 1 s
   "SV1401_close" : Bool = PLC SV1401_close AT %M0.7, 1 s
   "SV1401_open" : Bool = PLC SV1401_open AT %M0.6, 1 s
   "FP_Database_SV 1401" : String[254] = PLC FP_Database."SV 1401" AT %DB1.DBX776.0, 1 s
   "SV1402_ close" : Bool = PLC "SV1402_ close" AT %M1.7, 1 s
   "SV1402_open" : Bool = PLC SV1402_open AT %M1.6, 1 s
   "FP_Database_SV1402" : String[254] = PLC FP_Database.SV1402 AT %DB1.DBX1808.0, 1 s
   "FP_Database_SV1502" : String[254] = PLC FP_Database.SV1502 AT %DB1.DBX2066.0, 1 s
   "SV1501_close" : Bool = PLC SV1501_close AT %M1.1, 1 s
   "SV1501_open" : Bool = PLC SV1501_open AT %M1.0, 1 s
   "SV1502_close" : Bool = PLC SV1502_close AT %M2.1, 1 s
   "SV1502_open" : Bool = PLC SV1502_open AT %M2.0, 1 s
   "FP_Database_SV1601" : String[254] = PLC FP_Database.SV1601 AT %DB1.DBX1292.0, 1 s
   "SV1601_close" : Bool = PLC SV1601_close AT %M1.3, 1 s
   "SV1601_open" : Bool = PLC SV1601_open AT %M1.2, 1 s
   "SV1602_ close" : Bool = PLC "SV1602_ close" AT %M2.3, 1 s
   "SV1602_open" : Bool = PLC SV1602_open AT %M2.2, 1 s
   "FP_Database_SV1602" : String[254] = PLC FP_Database.SV1602 AT %DB1.DBX2324.0, 1 s
   "FP_Database_SV1702" : String[254] = PLC FP_Database.SV1702 AT %DB1.DBX2582.0, 1 s
   "SV1701_close" : Bool = PLC SV1701_close AT %M1.5, 1 s
   "SV1701_open" : Bool = PLC SV1701_open AT %M1.4, 1 s
   "SV1701" : Bool = PLC SV1701 AT %Q4.6, 1 s
   "FP_Database_SV1701" : String[254] = PLC FP_Database.SV1701 AT %DB1.DBX1550.0, 1 s
   "SV1702_close" : Bool = PLC SV1702_close AT %M2.5, 1 s
   "SV1702_open" : Bool = PLC SV1702_open AT %M2.4, 1 s
   "FP_Database_Pump_visibility_1(1)" : Bool = PLC FP_Database.Pump_visibility_1 AT %DB1.DBX0.0, 1 s
   "Alarms_fault" : Int AT %DB2.DBW0, 1 s
   "Level_real_140" : Real = PLC Level_real_140 AT %MD6, 1 s
   "Level_real_150" : Real = PLC Level_real_150 AT %MD10, 1 s
   "Level_real_160" : Real = PLC Level_real_160 AT %MD14, 1 s
   "Level_real_170" : Real = PLC Level_real_170 AT %MD18, 1 s
   "FP_Database_SV1501" : String[254] = PLC FP_Database.SV1501 AT %DB1.DBX1034.0, 1 s

discrete alarms
   1: 'Level transmitter 140 is not working / Cause of alarm: Level transmitter is out of range Corrective actions: Raise corrective order in maintenance system Consequence no action: No control or monitoring of the level in tank 140', class Acknowledgement, trigger "Alarms_fault" bit 8
   2: 'Level transmitter 150 is not working / Cause of alarm: Level transmitter is out of range Corrective actions: Raise corrective order in maintenance system Consequence no action: Overfill and overpressure', class Acknowledgement, trigger "Alarms_fault" bit 9
   3: 'Solenoid valve 1401 is failed to close / Cause of alarm: Solenoid valve is failed to close Corrective actions: Raise corrective order in maintenance system Consequence no action: Overfill and can not be controlled', class Errors, trigger "Alarms_fault" bit 10
   4: 'Solenoid valve 1502 is failed to open / Cause of alarm: Outlet solenoid valve is failed to open Corrective actions: Raise corrective order in maintenance system Consequence no action: cannot provide liquid to master tank', class Errors, trigger "Alarms_fault" bit 11
   5: 'Pump 771A is failed to start / Cause of alarm: Pump is failed to start Corrective actions: Raise corrective order in maintenance system Consequence no action: overfill and can not be controlled', class Errors, trigger "Alarms_fault" bit 12

analog alarms
   1: 'Low level alarm in tank 140', class Acknowledgement, trigger "Level_real_140"
   2: 'High level alarm in tank 140', class Acknowledgement, trigger "Level_real_140"
   3: 'Low level alarm in tank 150', class Acknowledgement, trigger "Level_real_150"
   4: 'High level alarm in tank 150', class Acknowledgement, trigger "Level_real_150"
   5: 'Low level alarm in tank 160', class Acknowledgement, trigger "Level_real_160"
   6: 'High level alarm in tank 160', class Acknowledgement, trigger "Level_real_160"
   7: 'Low level alarm in tank 170', class Acknowledgement, trigger "Level_real_170"
   8: 'High level alarm in tank 170', class Acknowledgement, trigger "Level_real_170"

screen "TANK_farm" 1024x767
   GraphicView "Graphic view_15" at 236,278 size 30x22; Picture "Graphic_35"
   GraphicView "Graphic view_18" at 242,163 size 18x119; Picture "Graphic_31"
   GraphicView "Graphic view_23" at 58,283 size 187x17; Picture "Graphic_30"
   GraphicView "Graphic view_5" at 418,431 size 180x136; Picture "Graphic_53"
   GraphicView "Graphic view_7" at 217,72 size 107x95; Picture "Graphic_53"
   GraphicView "Graphic view_4" at 436,74 size 107x95; Picture "Graphic_53"
   GraphicView "Graphic view_3" at 638,72 size 108x96; Picture "Graphic_53"
   GraphicView "Graphic view_32" at 198,626 size 285x14; Picture "Graphic_30"
   GraphicView "Graphic view_34" at 481,561 size 18x64; Picture "Graphic_31"
   GraphicView "Graphic view_35" at 513,562 size 18x63; Picture "Graphic_31"
   GraphicView "Graphic view_36" at 473,618 size 25x22; Picture "Graphic_37"
   GraphicView "Graphic view_33" at 514,619 size 26x23; Picture "Graphic_38"
   GraphicView "Graphic view_37" at 527,627 size 203x15; Picture "Graphic_30"
   GraphicView "Graphic view_22" at 652,275 size 25x24; Picture "Graphic_37"
   GraphicView "Graphic view_11" at 458,163 size 18x119; Picture "Graphic_31"
   GraphicView "Graphic view_21" at 476,283 size 187x17; Picture "Graphic_30"
   GraphicView "Graphic view_9" at 452,278 size 30x22; Picture "Graphic_35"
   GraphicView "Graphic view_17" at 660,164 size 18x118; Picture "Graphic_31"
   GraphicView "Graphic view_19" at 705,159 size 18x210; Picture "Graphic_31"
   GraphicView "Graphic view_20" at 697,358 size 25x24; Picture "Graphic_37"
   GraphicView "Graphic view_25" at 165,366 size 126x17; Picture "Graphic_30"
   GraphicView "Graphic view_28" at 283,361 size 30x22; Picture "Graphic_35"
   GraphicView "Graphic view_30" at 143,382 size 18x248; Picture "Graphic_31"
   GraphicView "Graphic view_29" at 144,367 size 25x24; Picture "Graphic_34"
   GraphicView "Graphic view_14" at 289,158 size 18x211; Picture "Graphic_31"
   GraphicView "Graphic view_16" at 258,283 size 203x17; Picture "Graphic_30"
   Group "Group" at 58,163 size 208x137; Picture "Graphic_35"
   GraphicView "Graphic view_40" at 242,190 size 45x41; Picture "Graphic_40"
      Appearance <- "SV1401"
   GraphicView "Graphic view_39" at 289,190 size 44x40; Picture "Graphic_40"
      Appearance <- "SV1402"
   GraphicView "Graphic view_10" at 507,158 size 18x210; Picture "Graphic_31"
   GraphicView "Graphic view_24" at 501,361 size 30x22; Picture "Graphic_35"
   GraphicView "Graphic view_27" at 306,366 size 202x17; Picture "Graphic_30"
   GraphicView "Graphic view_26" at 525,366 size 179x17; Picture "Graphic_30"
   GraphicView "Graphic view_13" at 458,190 size 45x40; Picture "Graphic_40"
      Appearance <- "SV1501"
   GraphicView "Graphic view_38" at 507,190 size 45x40; Picture "Graphic_40"
      Appearance <- "SV1502"
   GraphicView "Graphic view_8" at 660,192 size 45x38; Picture "Graphic_40"
      Appearance <- "SV1601"
   GraphicView "Graphic view_12" at 705,191 size 44x39; Picture "Graphic_40"
      Appearance <- "SV1602"
   GraphicView "Graphic view_44" at 25,282 size 42x43; Picture "Graphic_41"
   GraphicView "Graphic view_1" at 165,623 size 44x43; Picture "Graphic_41"
      Appearance <- "Pump770A"
   GraphicView "Graphic view_6" at 144,623 size 25x23; Picture "Graphic_38"
   GraphicView "Graphic view_46" at 718,616 size 44x43; Picture "Graphic_41"
      Appearance <- "Pump771A"
   GraphicView "Graphic view_47" at 608,594 size 56x50; Picture "Graphic_46"
   GraphicView "Graphic view_48" at 302,595 size 56x49; Picture "Graphic_46"
   Button "Button_1" at 251,41 size 74x33; TextOff 'Tank 140'
      on Click: ActivateScreen("TANK140", 0)
   Button "Button_2" at 469,42 size 74x32; TextOff 'Tank 150'
      on Click: ActivateScreen("TANK150", 0)
   Button "Button_3" at 671,38 size 77x33; TextOff 'Tank 160'
      on Click: ActivateScreen("TANK160", 0)
   Button "Button_4" at 476,401 size 74x30; TextOff 'Tank 170'
      on Click: ActivateScreen("TANK170", 0)
   Button "Button_5" at 879,84 size 96x32; TextOff 'MAIN'
      on Press: ActivateScreen("MAIN", 0)
   Circle "Circle_1" at 30,290 size 25x25
      Appearance <- "Pump100A"
   Circle "Circle_2" at 171,631 size 25x25
      Appearance <- "Pump770A"
   Circle "Circle_3" at 724,624 size 25x25
      Appearance <- "Pump771A"
   Rectangle "Rectangle_7" at 632,603 size 26x13
      Appearance <- "SV1702"
   Rectangle "Rectangle_8" at 324,603 size 27x13
      Appearance <- "SV1701"
   Rectangle "Rectangle_9" at 269,206 size 13x17
      Appearance <- "SV1401"
   Rectangle "Rectangle_10" at 315,206 size 13x17
      Appearance <- "SV1402"
   Rectangle "Rectangle_11" at 485,206 size 13x18
      Appearance <- "SV1501"
   Rectangle "Rectangle_12" at 534,207 size 13x17
      Appearance <- "SV1502"
   Rectangle "Rectangle_13" at 687,207 size 13x17
      Appearance <- "SV1601"
   Rectangle "Rectangle_14" at 730,207 size 13x17
      Appearance <- "SV1602"
   IOField "I/O field_1" at 233,117 size 82x29; FormatPattern 99999.9
      ProcessValue <- "Level_real_140"
   DateTimeField "Date/time field_1" at 830,14 size 188x26
   IOField "I/O field_2" at 449,117 size 82x29; FormatPattern 99999.9
      ProcessValue <- "Level_real_150"
   IOField "I/O field_3" at 652,112 size 82x29; FormatPattern 99999.9
      ProcessValue <- "Level_real_160"
   IOField "I/O field_4" at 453,495 size 110x29; FormatPattern 9999999.9
      ProcessValue <- "Level_real_170"
   IOField "I/O field_5" at 927,47 size 97x32; FormatPattern ????????
      ProcessValue <- "Current_user"
   TextField "Text field_12" at 836,51 size 80x22; Text 'Username'
   Button "Button_17" at 879,125 size 98x31; TextOff 'Alarms'; Authorization "Operate"
      on Press: ActivateScreen("Alarms", 0)
   Button "Button_26" at 879,165 size 98x31; TextOff 'Trends'; Authorization "Monitor"
      on Press: ActivateScreen("Trends", 0)
   TextField "Text field_13" at 192,47 size 23x56; Text 'LT 140'
   TextField "Text field_14" at 410,53 size 23x56; Text 'LT 150'
   TextField "Text field_15" at 613,47 size 23x56; Text 'LT 160'
   TextField "Text field_16" at 380,431 size 23x56; Text 'LT 170'
   GraphicView "Graphic view_51" at 792,49 size 38x32; Picture "Graphic_55"
   GraphicView "Graphic view_52" at 634,61 size 29x55; Picture "Graphic_56"
   GraphicView "Graphic view_53" at 437,62 size 29x55; Picture "Graphic_56"
   GraphicView "Graphic view_54" at 216,57 size 29x55; Picture "Graphic_56"
   GraphicView "Graphic view_55" at 424,416 size 29x55; Picture "Graphic_56"
   Rectangle "Rectangle_1" at 330,84 size 14x7
      Appearance <- "H_alarm_140"
   Rectangle "Rectangle_2" at 330,136 size 14x7
      Appearance <- "L_alarm_140"
   Button "Button_9" at 329,63 size 54x31; TextOff 'Text'
      on Click: function_efd93a16("High_alarm", 400, 200, -1, -1, 0)
   Button "Button_10" at 327,123 size 57x25; TextOff 'Text'
      on Click: function_efd93a16("Low_alarm", 400, 200, -1, -1, 1)
   GraphicView "Graphic view_2" at 351,73 size 20x21; Picture "in"
   GraphicView "Graphic view_31" at 346,128 size 20x21; Picture "in"
   Rectangle "Rectangle_3" at 547,92 size 14x7
      Appearance <- "H_alarm_150"
   Rectangle "Rectangle_4" at 547,144 size 14x7
      Appearance <- "L_alarm_150"
   Button "Button_6" at 544,78 size 54x31; TextOff 'Text'
      on Click: function_efd93a16("High_alarm", 400, 200, -1, -1, 0)
   Button "Button_7" at 544,134 size 57x25; TextOff 'Text'
      on Click: function_efd93a16("Low_alarm", 400, 200, -1, -1, 1)
   GraphicView "Graphic view_41" at 568,81 size 20x21; Picture "in"
   GraphicView "Graphic view_42" at 563,136 size 20x21; Picture "in"
   Rectangle "Rectangle_5" at 751,88 size 14x7
      Appearance <- "H_alarm_160"
   Rectangle "Rectangle_6" at 749,133 size 16x7
      Appearance <- "L_alarm_160"
   GraphicView "Graphic view_43" at 772,81 size 20x21; Picture "in"
   GraphicView "Graphic view_45" at 773,127 size 20x21; Picture "in"
   Rectangle "Rectangle_15" at 599,453 size 20x8
      Appearance <- "H_alarm_170"
   Rectangle "Rectangle_16" at 596,533 size 21x8
      Appearance <- "L_alarm_170"
   Button "Button_13" at 589,447 size 66x29; TextOff 'Text'
      on Click: function_efd93a16("High_alarm", 400, 200, -1, -1, 0)
   GraphicView "Graphic view_49" at 620,447 size 20x21; Picture "in"
   GraphicView "Graphic view_50" at 619,524 size 20x21; Picture "in"
   Button "Button_11" at 747,78 size 54x31; TextOff 'Text'
      on Click: function_efd93a16("High_alarm", 400, 200, -1, -1, 0)
   Button "Button_12" at 748,125 size 57x25; TextOff 'Text'
      on Click: function_efd93a16("Low_alarm", 400, 200, -1, -1, 1)
   Button "Button_14" at 597,440 size 54x31; TextOff 'Text'
      on Click: function_efd93a16("High_alarm", 400, 200, -1, -1, 0)
   Button "Button_31" at 592,524 size 57x25; TextOff 'Text'
      on Click: function_efd93a16("Low_alarm", 400, 200, -1, -1, 1)

Template "T1x0" 1024x767
   GraphicView "Graphic view_44" at 52,227 size 51x50; Picture "Graphic_41"
   GraphicView "Graphic view_1" at 770,324 size 53x46; Picture "Graphic_41"
   GraphicView "Graphic view_25" at 97,230 size 253x17; Picture "Graphic_30"
   GraphicView "Graphic view_2" at 497,338 size 285x19; Picture "Graphic_30"
   GraphicView "Template_Graphic view_1" at 599,316 size 48x41; Picture "Graphic_44"
   GraphicView "Template_Graphic view_2" at 213,206 size 48x41; Picture "Graphic_44"
   GraphicView "Graphic view_5" at 337,175 size 186x198; Picture "Graphic_53"
   GraphicView "Graphic view_55" at 349,160 size 29x55; Picture "Graphic_56"

screen "TANK150" 1024x767, template "T1x0"
   TextField "Text field_1" at 380,274 size 80x22; Text 'TANK 150'
   Button "Button_5" at 37,174 size 96x32; TextOff 'Pump 100A'
      on Press: SetBit("FP_Database_Pump_visibility_1(1)")
   Button "Button_6" at 753,280 size 96x32; TextOff 'Pump 770A'
      on Press: SetBit("FP_Database_Pump_visibility_2")
   Button "Button_11" at 193,170 size 96x32; TextOff 'SV 1501'
      on Press: SetBit("FP_Database_V_vis_1501")
   Button "Button_12" at 580,274 size 96x32; TextOff 'SV1502'
      on Press: SetBit("FP_Database_V_vis_1502")
   ScreenModuleView "Pump_valve_faceplate__2" at 507,371 size 176x153; ScreenModuleType ""
      Guid_{11997190-13903} <- "SV1502_close"
      Guid_{11997190-13901} <- "SV1502_open"
      Guid_{11997190-13905} <- "SV1502"
      Guid_{11997190-13907} <- "FP_Database_SV1502"
      Guid_{11997190-13897} <- "FP_Database_V_vis_1502"
   ScreenModuleView "Pump_valve_faceplate__3" at 174,298 size 173x151; ScreenModuleType ""
      Guid_{11997190-13903} <- "SV1501_close"
      Guid_{11997190-13901} <- "SV1501_open"
      Guid_{11997190-13905} <- "SV1501"
      Guid_{11997190-13897} <- "FP_Database_V_vis_1501"
      Guid_{11997190-13907} <- "FP_Database_SV1501"
   ScreenModuleView "Pump_valve_faceplate__4" at 3,299 size 166x151; ScreenModuleType ""
      Guid_{11997190-7773} <- "Pump100A"
      Guid_{11997190-7771} <- "Pump100A _stop"
      Guid_{11997190-7775} <- "FP_Database_Pump100A"
      Guid_{11997190-7769} <- "Pump100A _start"
      Guid_{11997190-7765} <- "FP_Database_Pump_visibility_1(1)"
   ScreenModuleView "Pump_valve_faceplate__1" at 713,381 size 152x146; ScreenModuleType ""
      Guid_{11997190-7773} <- "Pump770A"
      Guid_{11997190-7771} <- "Pump770A_stop"
      Guid_{11997190-7775} <- "FP_Database_Pump770"
      Guid_{11997190-7765} <- "FP_Database_Pump_visibility_2"
      Guid_{11997190-7769} <- "Pump770A _start"
   Bar "Bar_1" at 510,166 size 62x167; MinimumValue 0; MaximumValue 2500
      ProcessValue <- "Level_real_150"
   Circle "Circle_2" at 781,333 size 25x25
      Appearance <- "Pump770A"
   Circle "Circle_1" at 61,239 size 25x25
      Appearance <- "Pump100A"
   Rectangle "Rectangle_11" at 224,228 size 27x18
      Appearance <- "SV1501"
   Rectangle "Rectangle_12" at 610,339 size 27x17
      Appearance <- "SV1502"
   Button "Button_7" at 224,17 size 88x37; TextOff 'Tank 140'
      on Click: ActivateScreen("TANK140", 0)
   Button "Button_1" at 47,14 size 147x44; TextOff 'Tank Farm'
      on Click: ActivateScreen("TANK_farm", 0)
   Button "Button_3" at 331,18 size 89x36; TextOff 'Tank 160'
      on Click: ActivateScreen("TANK160", 0)
   Button "Button_4" at 436,18 size 84x37; TextOff 'Tank 170'
      on Click: ActivateScreen("TANK170", 0)
   Button "Button_8" at 75,69 size 101x34; TextOff 'Alarm page'
      on Click: ActivateScreen("Alarms", 0)
   DateTimeField "Date/time field_2" at 676,32 size 188x26
   IOField "I/O field_5" at 773,65 size 97x32; FormatPattern ????????
      ProcessValue <- "Current_user"
   TextField "Text field_12" at 682,69 size 80x22; Text 'Username'
   GraphicView "Graphic view_51" at 638,67 size 38x32; Picture "Graphic_55"

screen "TANK160" 1024x767, template "T1x0"
   TextField "Text field_1" at 377,270 size 80x22; Text 'TANK 160'
   TextField "Text field_3" at 544,178 size 15x22; Text 'Text'
   Button "Button_5" at 37,168 size 96x32; TextOff 'Pump 100A'
      on Press: SetBit("FP_Database_Pump_visibility_1(1)")
   Button "Button_6" at 753,280 size 96x32; TextOff 'Pump 770A'
      on Press: SetBit("FP_Database_Pump_visibility_2")
   Button "Button_11" at 193,170 size 96x32; TextOff 'SV 1601'
      on Press: SetBit("FP_Database_V_vis_1601")
   Button "Button_12" at 580,274 size 96x32; TextOff 'SV1602'
      on Press: SetBit("FP_Database_V_vis_1602")
   ScreenModuleView "Pump_valve_faceplate__2" at 516,382 size 167x146; ScreenModuleType ""
      Guid_{11997190-13903} <- "SV1602_ close"
      Guid_{11997190-13901} <- "SV1602_open"
      Guid_{11997190-13905} <- "SV1602"
      Guid_{11997190-13897} <- "FP_Database_V_vis_1602"
      Guid_{11997190-13907} <- "FP_Database_SV1602"
   ScreenModuleView "Pump_valve_faceplate__3" at 169,298 size 165x146; ScreenModuleType ""
      Guid_{11997190-13897} <- "FP_Database_V_vis_1601"
      Guid_{11997190-13907} <- "FP_Database_SV1601"
      Guid_{11997190-13903} <- "SV1601_close"
      Guid_{11997190-13901} <- "SV1601_open"
      Guid_{11997190-13905} <- "SV1601"
   ScreenModuleView "Pump_valve_faceplate__4" at 3,299 size 161x144; ScreenModuleType ""
      Guid_{11997190-7773} <- "Pump100A"
      Guid_{11997190-7771} <- "Pump100A _stop"
      Guid_{11997190-7775} <- "FP_Database_Pump100A"
      Guid_{11997190-7769} <- "Pump100A _start"
      Guid_{11997190-7765} <- "FP_Database_Pump_visibility_1(1)"
   ScreenModuleView "Pump_valve_faceplate__1" at 713,381 size 152x146; ScreenModuleType ""
      Guid_{11997190-7773} <- "Pump770A"
      Guid_{11997190-7771} <- "Pump770A_stop"
      Guid_{11997190-7775} <- "FP_Database_Pump770"
      Guid_{11997190-7765} <- "FP_Database_Pump_visibility_2"
      Guid_{11997190-7769} <- "Pump770A _start"
   Bar "Bar_1" at 510,166 size 62x167; MinimumValue 0; MaximumValue 3000
      ProcessValue <- "Level_real_160"
   Rectangle "Rectangle_13" at 224,229 size 27x16
      Appearance <- "SV1601"
   Rectangle "Rectangle_14" at 611,339 size 26x17
      Appearance <- "SV1602"
   Circle "Circle_1" at 61,239 size 25x25
      Appearance <- "Pump100A"
   Circle "Circle_2" at 780,333 size 25x25
      Appearance <- "Pump770A"
   Button "Button_2" at 229,18 size 88x37; TextOff 'Tank 140'
      on Click: ActivateScreen("TANK140", 0)
   Button "Button_1" at 47,14 size 147x44; TextOff 'Tank Farm'
      on Click: ActivateScreen("TANK_farm", 0)
   Button "Button_4" at 331,18 size 89x36; TextOff 'Tank 160'
      on Click: ActivateScreen("TANK160", 0)
   Button "Button_7" at 436,18 size 84x37; TextOff 'Tank 170'
      on Click: ActivateScreen("TANK170", 0)
   Button "Button_8" at 75,69 size 101x34; TextOff 'Alarm page'
      on Click: ActivateScreen("Alarms", 0)
   DateTimeField "Date/time field_2" at 676,32 size 188x26
   IOField "I/O field_5" at 773,65 size 97x32; FormatPattern ????????
      ProcessValue <- "Current_user"
   TextField "Text field_12" at 682,69 size 80x22; Text 'Username'
   GraphicView "Graphic view_51" at 638,67 size 38x32; Picture "Graphic_55"

screen "TANK170" 1024x767, template "T1x0"
   TextField "Text field_1" at 389,280 size 80x22; Text 'TANK 170'
   Button "Button_5" at 37,170 size 96x32; TextOff 'Pump 770A'
      on Press: SetBit("FP_Database_Pump_visibility_2")
   Button "Button_6" at 753,280 size 96x32; TextOff 'Pump 771A'
      on Press: SetBit("FP_Database_Pump_visibility_3")
   Button "Button_11" at 193,170 size 96x32; TextOff 'SV 1701'
      on Press: SetBit("FP_Database_V_vis_1701")
   Button "Button_12" at 580,274 size 96x32; TextOff 'SV1702'
      on Press: SetBit("FP_Database_V_vis_1702")
   ScreenModuleView "Pump_valve_faceplate__2" at 516,382 size 167x146; ScreenModuleType ""
      Guid_{11997190-13897} <- "FP_Database_V_vis_1702"
      Guid_{11997190-13907} <- "FP_Database_SV1702"
      Guid_{11997190-13903} <- "SV1702_close"
      Guid_{11997190-13901} <- "SV1702_open"
      Guid_{11997190-13905} <- "SV1702"
   ScreenModuleView "Pump_valve_faceplate__3" at 174,297 size 160x147; ScreenModuleType ""
      Guid_{11997190-13903} <- "SV1701_close"
      Guid_{11997190-13901} <- "SV1701_open"
      Guid_{11997190-13905} <- "SV1701"
      Guid_{11997190-13907} <- "FP_Database_SV1701"
      Guid_{11997190-13897} <- "FP_Database_V_vis_1701"
   ScreenModuleView "Pump_valve_faceplate__5" at 10,298 size 157x146; ScreenModuleType ""
      Guid_{11997190-7773} <- "Pump770A"
      Guid_{11997190-7771} <- "Pump770A_stop"
      Guid_{11997190-7775} <- "FP_Database_Pump770"
      Guid_{11997190-7765} <- "FP_Database_Pump_visibility_2"
      Guid_{11997190-7769} <- "Pump770A _start"
   Bar "Bar_1" at 510,166 size 62x167; MinimumValue 0; MaximumValue 10000
      ProcessValue <- "Level_real_170"
   Circle "Circle_2" at 62,239 size 25x25
      Appearance <- "Pump770A"
   Rectangle "Rectangle_8" at 223,229 size 29x16
      Appearance <- "SV1701"
   Rectangle "Rectangle_7" at 610,339 size 27x17
      Appearance <- "SV1702"
   Circle "Circle_3" at 781,334 size 25x25
      Appearance <- "Pump771A"
   ScreenModuleView "Pump_valve_faceplate__4" at 698,384 size 151x143; ScreenModuleType ""
      Guid_{11997190-7765} <- "FP_Database_Pump_visibility_3"
      Guid_{11997190-7769} <- "Pump771A _start"
      Guid_{11997190-7773} <- "Pump771A"
      Guid_{11997190-7771} <- "Pump771A _stop"
      Guid_{11997190-7775} <- "FP_Database_Pump771"
   Button "Button_1" at 47,14 size 147x44; TextOff 'Tank Farm'
      on Click: ActivateScreen("TANK_farm", 0)
   Button "Button_2" at 317,14 size 88x37; TextOff 'Tank 150'
      on Click: ActivateScreen("TANK150", 0)
   Button "Button_3" at 421,16 size 89x36; TextOff 'Tank 160'
      on Click: ActivateScreen("TANK160", 0)
   Button "Button_8" at 75,69 size 101x34; TextOff 'Alarm page'
      on Click: ActivateScreen("Alarms", 0)
   DateTimeField "Date/time field_2" at 676,32 size 188x26
   IOField "I/O field_5" at 773,65 size 97x32; FormatPattern ????????
      ProcessValue <- "Current_user"
   TextField "Text field_12" at 682,69 size 80x22; Text 'Username'
   GraphicView "Graphic view_51" at 638,67 size 38x32; Picture "Graphic_55"
   Button "Button_7" at 214,14 size 88x37; TextOff 'Tank 140'
      on Click: ActivateScreen("TANK140", 0)

screen "MAIN" 1024x767
   Button "Button_1" at 298,21 size 96x32; TextOff 'Login'
      on Press: function_a2a04561()
   Button "Button_2" at 467,21 size 96x32; TextOff 'Logoff'
      on Press: function_f23ef4c9()
   Button "Button_3" at 722,114 size 99x32; TextOff 'Tank farm'; Authorization "Operate"
      on Press: ActivateScreen("TANK_farm", 0)
   IOField "I/O field_1" at 385,63 size 227x32; FormatPattern ????????
      ProcessValue <- "Current_user"
   UserView "User view_1" at 180,114 size 480x240
   TextField "Text field_1" at 218,64 size 144x22; Text 'Current username:'
   Button "Button_4" at 723,155 size 98x31; TextOff 'Alarms'; Authorization "Operate"
      on Press: ActivateScreen("Alarms", 0)
   Button "Button_5" at 723,195 size 98x31; TextOff 'Trends'; Authorization "Operate"
      on Press: ActivateScreen("Trends", 0)

PopupScreen "High_alarm" 270x170
   Button "Button_1" at 233,2 size 26x22; TextOff 'X'
      on Click: function_efd93a16("High_alarm", 0, 0, 0, -1, 1)
   GraphicView "Graphic view_1" at 12,36 size 247x116; Picture "high_1"

PopupScreen "Low_alarm" 270x170
   Button "Button_1" at 234,1 size 26x22; TextOff 'X'
      on Click: function_efd93a16("Low_alarm", 0, 0, 0, -1, 1)
   GraphicView "Graphic view_1" at 7,30 size 247x127; Picture "low_1"

screen "TANK140" 1024x767, template "T1x0"
   Button "Button_1" at 47,14 size 147x44; TextOff 'Tank Farm'
      on Click: ActivateScreen("TANK_farm", 0)
   Button "Button_2" at 220,17 size 88x37; TextOff 'Tank 150'
      on Click: ActivateScreen("TANK150", 0)
   Button "Button_3" at 331,18 size 89x36; TextOff 'Tank 160'
      on Click: ActivateScreen("TANK160", 0)
   Button "Button_4" at 436,18 size 84x37; TextOff 'Tank 170'
      on Click: ActivateScreen("TANK170", 0)
   Button "Button_6" at 753,280 size 96x32; TextOff 'Pump 770A'
      on Press: SetBit("FP_Database_Pump_visibility_2")
   Button "Button_10" at 928,685 size 96x32; TextOff 'Pump 100A'
      on Press: SetBit("FP_Database_Pump_visibility_1(1)")
   Button "Button_11" at 193,170 size 96x32; TextOff 'SV 1401'
      on Click: SetBit("FP_Database_V_vis_1401")
   Button "Button_12" at 580,274 size 96x32; TextOff 'SV1402'
      on Press: SetBit("FP_Database_V_vis_1402")
   ScreenModuleView "Pump_valve_faceplate__1" at 697,380 size 168x147; ScreenModuleType ""
      Guid_{11997190-7765} <- "FP_Database_Pump_visibility_2"
      Guid_{11997190-7769} <- "Pump770A _start"
      Guid_{11997190-7773} <- "Pump770A"
      Guid_{11997190-7771} <- "Pump770A_stop"
      Guid_{11997190-7775} <- "FP_Database_Pump770"
   ScreenModuleView "Pump_valve_faceplate__2" at 508,380 size 173x146; ScreenModuleType ""
      Guid_{11997190-13897} <- "FP_Database_V_vis_1402"
      Guid_{11997190-13903} <- "SV1402_ close"
      Guid_{11997190-13901} <- "SV1402_open"
      Guid_{11997190-13905} <- "SV1402"
      Guid_{11997190-13907} <- "FP_Database_SV1402"
   ScreenModuleView "Pump_valve_faceplate__3" at 178,295 size 161x152; ScreenModuleType ""
      Guid_{11997190-13897} <- "FP_Database_V_vis_1401"
      Guid_{11997190-13903} <- "SV1401_close"
      Guid_{11997190-13901} <- "SV1401_open"
      Guid_{11997190-13905} <- "SV1401"
      Guid_{11997190-13907} <- "FP_Database_SV 1401"
   ScreenModuleView "Pump_valve_faceplate__4" at 3,295 size 158x153; ScreenModuleType ""
      Guid_{11997190-7769} <- "Pump100A _start"
      Guid_{11997190-7773} <- "Pump100A"
      Guid_{11997190-7771} <- "Pump100A _stop"
      Guid_{11997190-7775} <- "FP_Database_Pump100A"
      Guid_{11997190-7765} <- "FP_Database_Pump_visibility_1(1)"
   Button "Button_5" at 45,176 size 95x32; TextOff 'Pump'
      on Click: SetBit("FP_Database_Pump_visibility_1(1)")
   TextField "Text field_1" at 380,274 size 80x22; Text 'TANK 140'
   Bar "Bar_1" at 510,166 size 62x167; MinimumValue 0; MaximumValue 1500
      ProcessValue <- "Level_real_140"
   Circle "Circle_1" at 61,239 size 25x25
      Appearance <- "Pump100A"
   Rectangle "Rectangle_9" at 223,229 size 29x17
      Appearance <- "SV1401"
   Rectangle "Rectangle_10" at 609,338 size 27x18
      Appearance <- "SV1402"
   Circle "Circle_2" at 780,333 size 25x25
      Appearance <- "Pump770A"
   Button "Button_8" at 75,69 size 101x34; TextOff 'Alarm page'
      on Click: ActivateScreen("Alarms", 0)
   DateTimeField "Date/time field_2" at 676,32 size 188x26
   IOField "I/O field_5" at 773,65 size 97x32; FormatPattern ????????
      ProcessValue <- "Current_user"
   TextField "Text field_12" at 682,69 size 80x22; Text 'Username'
   GraphicView "Graphic view_51" at 638,67 size 38x32; Picture "Graphic_55"

screen "Alarms" 1024x767
   Button "Button_1" at 744,172 size 145x44; TextOff 'Main'
      on Click: ActivateScreen("MAIN", 0)
   DateTimeField "Date/time field_1" at 698,85 size 247x32
   Button "Button_2" at 745,224 size 147x47; TextOff 'Tank Farm'
      on Click: ActivateScreen("TANK_farm", 0)
   AlarmView "Alarm view_1" at 43,85 size 600x300
   TextField "Text field_1" at 229,14 size 174x37; Text 'Alarms Page'
   IOField "I/O field_5" at 833,130 size 97x32; FormatPattern ????????
      ProcessValue <- "Current_user"
   TextField "Text field_12" at 742,134 size 80x22; Text 'Username'
   GraphicView "Graphic view_51" at 698,132 size 38x32; Picture "Graphic_55"

screen "Trends" 1024x767
   TrendView "Trend view_1" at 43,73 size 745x628
   GraphicView "Graphic view_1" at 808,616 size 177x79; Picture "Capture4"
   Button "Button_1" at 854,206 size 145x44; TextOff 'Main'
      on Click: ActivateScreen("MAIN", 0)
   Button "Button_2" at 852,269 size 147x47; TextOff 'Tank Farm'
      on Click: ActivateScreen("TANK_farm", 0)
   TextField "Text field_1" at 816,586 size 59x22; Text 'Legend'
   TextField "Text field_2" at 271,13 size 185x39; Text 'Trends Page'
   DateTimeField "Date/time field_1" at 830,125 size 188x26
   IOField "I/O field_5" at 927,158 size 97x32; FormatPattern ????????
      ProcessValue <- "Current_user"
   TextField "Text field_12" at 836,162 size 80x22; Text 'Username'
   GraphicView "Graphic view_51" at 792,160 size 38x32; Picture "Graphic_55"

scheduled task "ChangeUsertask"
   on Action: function_f41c6f6c("Current_user"); function_de9337da(); function_e1ab61de("Gruop_number")
*)

(* ===== HMI "HMI_RT_1" =====
system functions are stored by id; their names below are inferred from use

text list "Status": 0 'OFF'; 1 'ON'

ScreenModuleEditorView "Pump_valve_faceplate_" 640x480
   Rectangle "Rectangle_1" at 140,25 size 192x176
      Visibility <- "FP_visibility"
   Button "Button_5" at 311,26 size 21x25; TextOff 'X'
      on Click: ResetBit("FP_visibility")
      Visibility <- "FP_visibility"
   Button "Button_6" at 149,157 size 76x30; TextOff 'Start'
      on Release: ResetBit("Pump_start")
      on Press: SetBit("Pump_start")
      Visibility <- "FP_visibility"
      ProcessValue <- "Pump_start"
   Button "Button_7" at 241,156 size 86x30; TextOff 'Stop'
      on Release: ResetBit("Pump_stop")
      on Press: SetBit("Pump_stop")
      Visibility <- "FP_visibility"
      ProcessValue <- "Pump_stop"
   SymbolicIOField "Symbolic I/O field_1" at 244,100 size 68x32; TextOn '1'; TextOff '0'; TextList "Status"
      ProcessValue <- "Pump_status"
      Visibility <- "FP_visibility"
   TextField "Text field_5" at 161,107 size 64x22; Text 'STATUS'
      Visibility <- "FP_visibility"
   IOField "I/O field_1" at 156,34 size 144x39; FormatPattern ????????
      ProcessValue <- "PumpTagNumber"
      Visibility <- "FP_visibility"
*)

(* ===== HMI "HMI_RT_1" =====
system functions are stored by id; their names below are inferred from use

text list "Status": 0 'Closed'; 1 'Opened'

ScreenModuleEditorView "Pump_valve_faceplate_" 640x480
   Rectangle "Rectangle_1" at 140,25 size 192x176
      Visibility <- "FP_valve"
   Button "Button_5" at 311,26 size 21x25; TextOff 'X'
      on Click: ResetBit("FP_valve")
      Visibility <- "FP_valve"
   Button "Button_6" at 149,157 size 76x30; TextOff 'Open'
      on Release: ResetBit("Valve_open")
      on Press: SetBit("Valve_open")
      Visibility <- "FP_valve"
      ProcessValue <- "Valve_open"
   Button "Button_7" at 241,156 size 86x30; TextOff 'Close'
      on Release: ResetBit("Valve_close")
      on Press: SetBit("Valve_close")
      Visibility <- "FP_valve"
      ProcessValue <- "Valve_close"
   SymbolicIOField "Symbolic I/O field_1" at 237,99 size 87x32; TextOn '1'; TextOff '0'; TextList "Status"
      Visibility <- "FP_valve"
      ProcessValue <- "Valve_status"
   TextField "Text field_5" at 161,107 size 64x22; Text 'STATUS'
      Visibility <- "FP_valve"
   IOField "I/O field_1" at 153,35 size 147x45; FormatPattern ????????
      Visibility <- "FP_valve"
      ProcessValue <- "ValveTagNumber"
*)